# EPICS substitutions: ipimbLib/Db/ipimb_iocAdmin.substitutions
#==============================================================================
#
# Abs:  IOC Administration Records
#
# Name: iocAdmin.substitutions
#
#==============================================================================
#
file iocSoft.db
{
	pattern
	{ IOCNAME }
	{ $(IOC)  }
}
